PROGRAM MAIN
VAR
	tonWritePersistent						: TON;
	fbPersistent 							: FB_WritePersistentData;
END_VAR

tonWritePersistent(IN:= NOT tonWritePersistent.Q, PT:= T#1M, Q=> , ET=> );		// Zapis persistentow
fbPersistent(PORT:= 851, START:= tonWritePersistent.Q);							// Zapis persistentow
P_EventsHS();

END_PROGRAM

(* stored: Version 1.1.0.1, ProductVersion 3.1.4022.12
   POU MAIN: Id {f4454d12-77f9-4a4f-9a67-d98ee49ff4c1}, SpecialFunc None *)
